// TIA Portal V19 export
TYPE "lexchangetray_typeUnEmn_signalTM_Monitor"
// Type: Bool
// stored: Access Published
   STRUCT
      simulationed : Bool;
   END_STRUCT;
END_TYPE
